Omron CX-Programmer project NewProject (CX-Programmer 9.72)

# PLC NewPLC1: CS1G-H CPU42

## Global symbols (name address type ; comment)
T0001 BOOL  ; Timer vervanging 5b6

## Program NewProgram1 (cyclic task 0)

### Section Section1

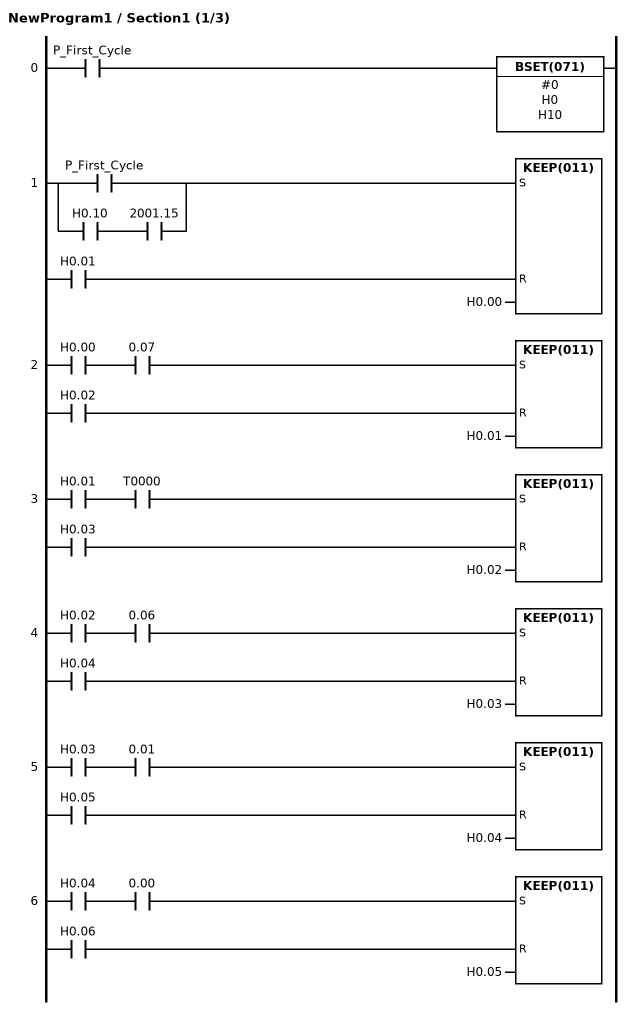
; rung 0
LD P_First_Cycle
BSET(071) #0 H0 H10
; rung 1
LD P_First_Cycle
LD H0.10
AND 2001.15
ORLD
LD H0.01
KEEP(011) H0.00
; rung 2
LD H0.00
AND 0.07
LD H0.02
KEEP(011) H0.01
; rung 3
LD H0.01
AND T0000
LD H0.03
KEEP(011) H0.02
; rung 4
LD H0.02
AND 0.06
LD H0.04
KEEP(011) H0.03
; rung 5
LD H0.03
AND 0.01
LD H0.05
KEEP(011) H0.04
; rung 6
LD H0.04
AND 0.00
LD H0.06
KEEP(011) H0.05

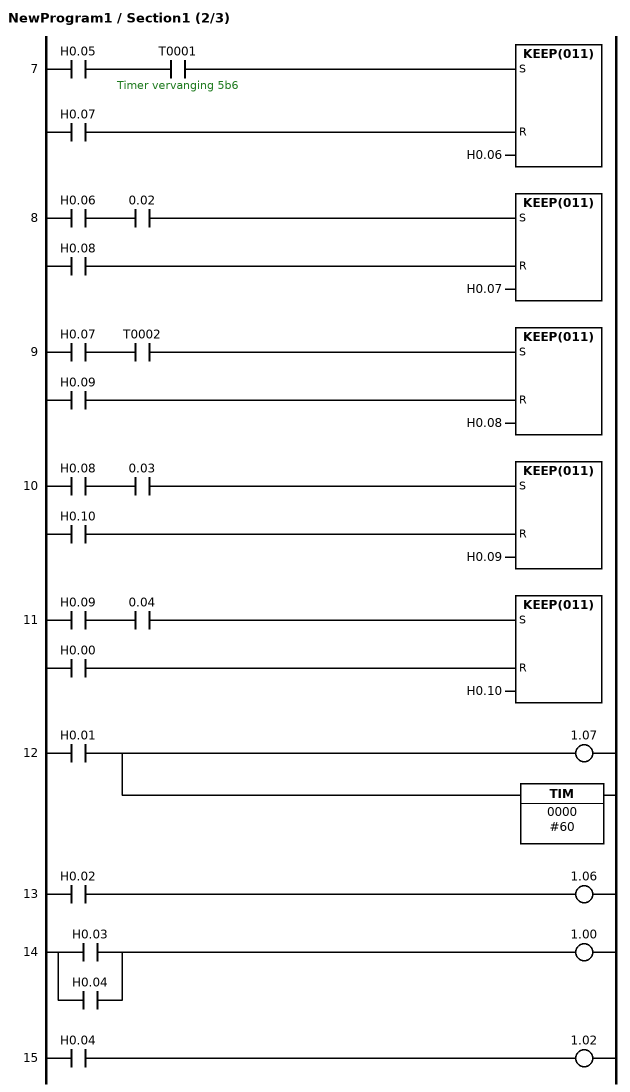
; rung 7
LD H0.05
AND T0001  ; Timer vervanging 5b6
LD H0.07
KEEP(011) H0.06
; rung 8
LD H0.06
AND 0.02
LD H0.08
KEEP(011) H0.07
; rung 9
LD H0.07
AND T0002
LD H0.09
KEEP(011) H0.08
; rung 10
LD H0.08
AND 0.03
LD H0.10
KEEP(011) H0.09
; rung 11
LD H0.09
AND 0.04
LD H0.00
KEEP(011) H0.10
; rung 12
LD H0.01
OUT 1.07
TIM 0000 #60
; rung 13
LD H0.02
OUT 1.06
; rung 14
LD H0.03
OR H0.04
OUT 1.00
; rung 15
LD H0.04
OUT 1.02

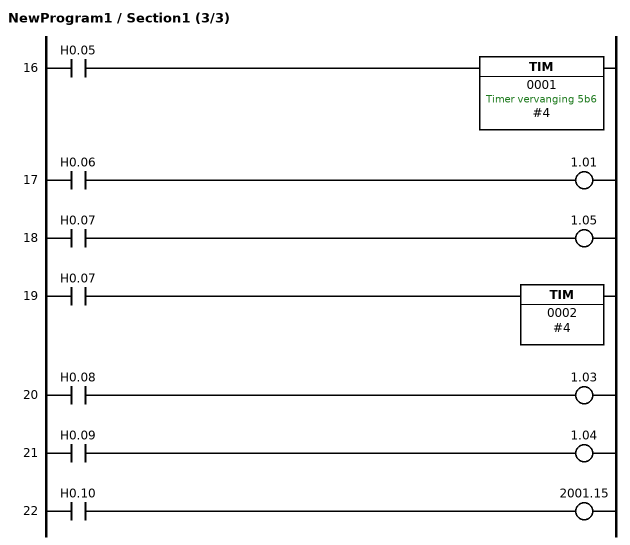
; rung 16
LD H0.05
TIM 0001 #4  ; Timer vervanging 5b6
; rung 17
LD H0.06
OUT 1.01
; rung 18
LD H0.07
OUT 1.05
; rung 19
LD H0.07
TIM 0002 #4
; rung 20
LD H0.08
OUT 1.03
; rung 21
LD H0.09
OUT 1.04
; rung 22
LD H0.10
OUT 2001.15

### Section END
; rung 0
END(001)